// TIA Portal V20 export
DATA_BLOCK "MP102"   // DB304
// stored: MemoryReserve 100
   VAR
      "LOWER 2-1 HEATER POWER TRIPPED E6168CB" : Bool;
      "LOWER 2-2 HEATER POWER TRIPPED E6174CB" : Bool;
      "LOWER 2-3 HEATER POWER TRIPPED E6180CB" : Bool;
      "VISION LIGHT CONTROLLER POWER STRIP OUTLET POWER TRIPPED E7184CB" : Bool;
      "120VAC CONTROL POWER TR PRIMARY TRIPPED E7100CB" : Bool;
      "120VAC CONTROL POWER TR SECONDARY TRIPPED E7110CB" : Bool;
      "CONTROL POWER ON TRIPPED E7116CB" : Bool;
      "MOTOR PANEL CONTROL POWER TRIPPED E7154CB" : Bool;
      "WEIGHT TESTER POWER STRIP OUTLET POWER TRIPPED E7160CB" : Bool;
      "VISION MONITOR & MCU POWER STRIP OUTLET POWER TRIPPED E7166CB" : Bool;
      "QR LASER MARKING TRIPPED E7172CB" : Bool;
      "HI-POT TESTER POWER STRIP OUTLET POWER TRIPPED E7178CB" : Bool;
      "FFU-1 POWER TRIPPED E7222CB" : Bool;
      "UPPER 1-1 TEMPERATURE CONTROLLER POWER TRIPPED E5206CB" : Bool;
      "UPPER 1-2 TEMPERATURE CONTROLLER POWER TRIPPED E5212CB" : Bool;
      "LOWER 1-1 TEMPERATURE CONTROLLER POWER TRIPPED E5218CB" : Bool;
      "LOWER 1-2 TEMPERATURE CONTROLLER POWER TRIPPED E5224CB" : Bool;
      "LOWER 1-3 TEMPERATURE CONTROLLER POWER TRIPPED E5230CB" : Bool;
      "UPPER 2-1 TEMPERATURE CONTROLLER POWER TRIPPED E6206CB" : Bool;
      "UPPER 2-2 TEMPERATURE CONTROLLER POWER TRIPPED E6212CB" : Bool;
      "LOWER 2-1 TEMPERATURE CONTROLLER POWER TRIPPED E6218CB" : Bool;
      "LOWER 2-2 TEMPERATURE CONTROLLER POWER TRIPPED E6224CB" : Bool;
      "LOWER 2-3 TEMPERATURE CONTROLLER POWER TRIPPED E6230CB" : Bool;
      SPARE : Bool;
      "CONTROL POWER SMPS DC OK E8104PWS" : Bool;
      "ET200MP I/O OUTPUT POWER TRIPPED E8154CB" : Bool;
      "JUNCTION BOX CONTROL POWER TRIPPED E8180CB" : Bool;
      "CLASS 2 SMPS POWER TRIPPED E8204CB" : Bool;
      "CLASS 2 SMPS MONITORING E8206PWS" : Bool;
      "ET200ECO PN-1 POWER TRIPPED E8220CB" : Bool;
      "ET200ECO PN-2 POWER TRIPPED E8224CB" : Bool;
      "ET200ECO PN-3 POWER TRIPPED E8228CB" : Bool;
   END_VAR
BEGIN
END_DATA_BLOCK
